// TIA Portal V17 export
// export: Created 2025-03-10T13:11:57.9169083Z, ExportSetting WithDefaults, DisplayName Totally Integrated Automation Portal, DisplayVersion V17 Update 8, DisplayName TIA Portal Openness, DisplayVersion V17 Update 8, DisplayName TIA Portal Version Control Interface, DisplayVersion V17, DisplayName SINAMICS Startdrive Advanced, DisplayVersion V17 SP2, DisplayName SINAMICS Startdrive G110M, G120, G120C, G120D, G120P, G115D, DisplayVersion V17 SP2, DisplayName SINAMICS Startdrive G130, G150, S120, S150, SINAMICS MV, S210, DisplayVersion V17 SP2, DisplayName STEP 7 Professional, DisplayVersion V17 Update 8, DisplayName SINUMERIK ONE STEP 7 Toolbox, DisplayVersion V17 Update 12, DisplayName SINUMERIK 840D sl STEP 7 Toolbox, DisplayVersion V17 Update 12, DisplayName STEP 7 Safety, DisplayVersion V17 Update 6, DisplayName WinCC Advanced, DisplayVersion V17 Update 8
TYPE "LBP_typeMcp483AdditionalOutput"
TITLE = MCP 483 image / Imagen de MCP 483 / MCP 483 Abbild
// Additional output image of MCP 483 / Imagen de salida adicional de MCP 483 / Zusätzliches Ausgangsabbild von MCP 483
// stored: IsFailsafeCompliant false
   STRUCT
      reserved1 : Byte;
      optionalKey1 : Bool;   // KT-OUT1,
      optionalKey2 : Bool;   // KT-OUT2
      optionalKey3 : Bool;   // KT-OUT3
      optionalKey4 : Bool;   // KT-OUT4
      optionalKey5 : Bool;   // KT-OUT5
      optionalKey6 : Bool;   // KT-OUT6
      reserved16 : Bool;
      reserved17 : Bool;
   END_STRUCT;
END_TYPE
